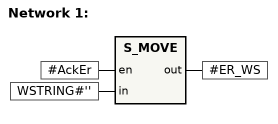
   IF #AckEr THEN #ER_WS := WSTRING#''; END_IF;
END_REGION

REGION Network 2 (SCL)

   #para_Artlimits := #para_in;
   #ER := false;
   IF #artLimfwd < #artLimRev THEN
       #ER_WS := #ER_WSlimfwdrev;
       #ER := true;
   ELSIF #UseArtLimitw THEN
       #para_Artlimits.pos_lim_fwd_USER := MIN(IN1 := #para_in.pos_lim_fwd_USER, IN2 := #artLimfwd);
       #para_Artlimits.pos_lim_rev_USER := MAX(IN1 := #para_in.pos_lim_rev_USER, IN2 := #artLimRev);
   END_IF;
END_REGION
END_FUNCTION_BLOCK

FUNCTION_BLOCK "axis_manager"   // FB25, FBD
{ S7_Optimized_Access := 'TRUE' }
VERSION : 0.1
// stored: AutoNumber true, IsIECCheckEnabled false, IsRetainMemResEnabled false, MemoryReserve 100, SetENOAutomatically false, UDAEnableTagReadback false
   VAR_INPUT
      allowed : Bool;
      targetUnison : Real;
      targetHome : Real;
      targetStep : Real;
      bSoftStop : Bool;
      bHome : Bool;
      hbStepPlus : Bool;
      hbStepMinus : Bool;
      bFwd : Bool;
      bRev : Bool;
      Params : "typeMotPara";
      ExecUni : Bool;
      theseAreDoors : Bool;
      xOverrideLOCAL : Bool;
      POS : Real;
   END_VAR
   VAR_OUTPUT
      team_unison : Bool;
      team_free : Bool;
      team_override : Bool;
      Desk_slowly : Bool;
      yaSpeedManual : Real;
      yaSpeedAuto : Real;
      m_auto : Bool;
      m_man : Bool;
      au_execute : Bool;
      aut_target : Real;
      OVERRIDE : Bool;
      ExecutingManuverFreeMode : Bool;
   END_VAR
   VAR
      st_Fwd : Bool;
      st_Rev : Bool;
      st_speed_slow_or_fast_negative : Real;
      aman_sel_target_Instance { S7_SetPoint := 'True'} : "aman_sel_target";
   END_VAR
   VAR_TEMP
      st_speedManual_slow_or_fast : Real;
      SpeedBlind : Real;
      stSpeedManualSlow : Real;
      Speed_autoSlow : Real;
   END_VAR
BEGIN

REGION Network 1
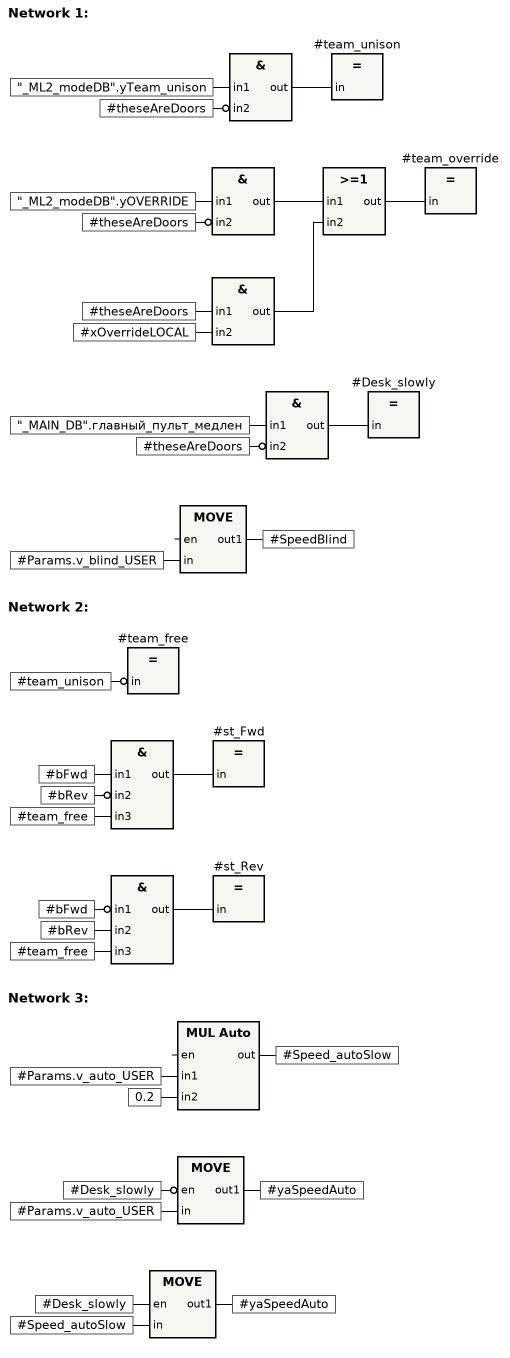
   #team_unison := "_ML2_modeDB".yTeam_unison AND NOT #theseAreDoors;
   #team_override := ("_ML2_modeDB".yOVERRIDE AND NOT #theseAreDoors) OR (#theseAreDoors AND #xOverrideLOCAL);
   #Desk_slowly := "_MAIN_DB".главный_пульт_медлен AND NOT #theseAreDoors;
   #SpeedBlind := #Params.v_blind_USER;
END_REGION

REGION Network 2
   #team_free := NOT #team_unison;
   #st_Fwd := #bFwd AND NOT #bRev AND #team_free;
   #st_Rev := NOT #bFwd AND #bRev AND #team_free;
END_REGION

REGION Network 3
   #Speed_autoSlow := #Params.v_auto_USER * 0.2;
   IF NOT #Desk_slowly THEN #yaSpeedAuto := #Params.v_auto_USER; END_IF;
   IF #Desk_slowly THEN #yaSpeedAuto := #Speed_autoSlow; END_IF;
END_REGION

REGION Network 4
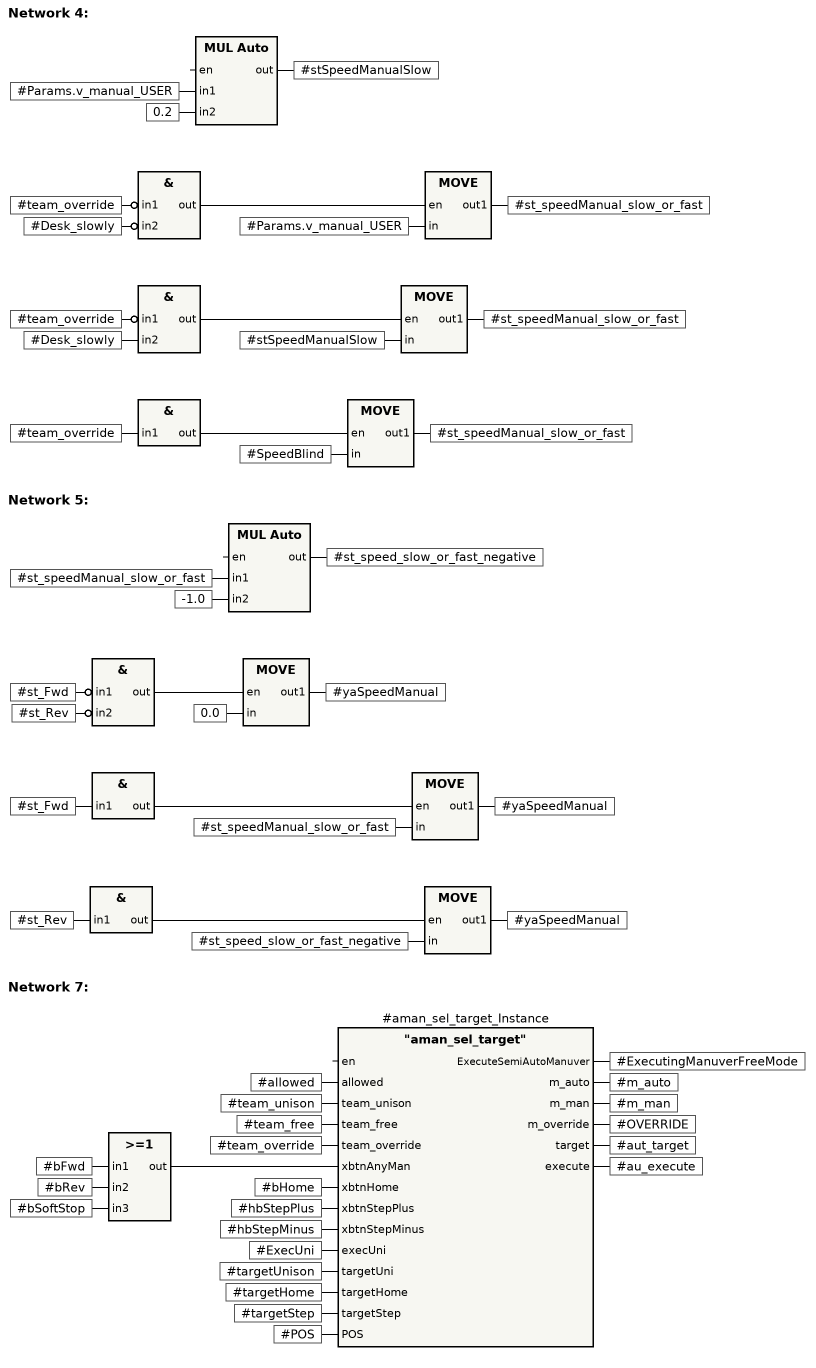
   #stSpeedManualSlow := #Params.v_manual_USER * 0.2;
   IF NOT #team_override AND NOT #Desk_slowly THEN
       #st_speedManual_slow_or_fast := #Params.v_manual_USER;
   END_IF;
   IF NOT #team_override AND #Desk_slowly THEN #st_speedManual_slow_or_fast := #stSpeedManualSlow; END_IF;
   IF #team_override THEN #st_speedManual_slow_or_fast := #SpeedBlind; END_IF;
END_REGION

REGION Network 5
   #st_speed_slow_or_fast_negative := #st_speedManual_slow_or_fast * (-1.0);
   IF NOT #st_Fwd AND NOT #st_Rev THEN #yaSpeedManual := 0.0; END_IF;
   IF #st_Fwd THEN #yaSpeedManual := #st_speedManual_slow_or_fast; END_IF;
   IF #st_Rev THEN #yaSpeedManual := #st_speed_slow_or_fast_negative; END_IF;
END_REGION

REGION Network 7
   #aman_sel_target_Instance(allowed := #allowed,   // "aman_sel_target"
                           team_unison := #team_unison,
                           team_free := #team_free,
                           team_override := #team_override,
                           xbtnAnyMan := #bFwd OR #bRev OR #bSoftStop,
                           xbtnHome := #bHome,
                           xbtnStepPlus := #hbStepPlus,
                           xbtnStepMinus := #hbStepMinus,
                           execUni := #ExecUni,
                           targetUni := #targetUnison,
                           targetHome := #targetHome,
                           targetStep := #targetStep,
                           POS := #POS,
                           ExecuteSemiAutoManuver => #ExecutingManuverFreeMode,
                           m_auto => #m_auto,
                           m_man => #m_man,
                           m_override => #OVERRIDE,
                           target => #aut_target,
                           execute => #au_execute);
END_REGION
END_FUNCTION_BLOCK

FUNCTION_BLOCK "aman_sel_target"   // FB58, FBD
{ S7_Optimized_Access := 'TRUE' }
VERSION : 0.1
// stored: AutoNumber true, IsIECCheckEnabled false, IsRetainMemResEnabled false, MemoryReserve 100, SetENOAutomatically false, UDAEnableTagReadback false
   VAR_INPUT
      allowed : Bool;
      team_unison : Bool;
      team_free : Bool;
      team_override : Bool;
      xbtnAnyMan : Bool;
      xbtnHome : Bool;
      xbtnStepPlus : Bool;
      xbtnStepMinus : Bool;
      execUni : Bool;
      targetUni : Real;
      targetHome : Real;
      targetStep : Real;
      POS : Real;
   END_VAR
   VAR_OUTPUT
      ExecuteSemiAutoManuver : Bool;
      m_auto : Bool;
      m_man : Bool;
      m_override : Bool;
      target : Real;
      execute : Bool;
   END_VAR
   VAR
      auto_allowed : Bool;
      anyBtn : Bool;
      xbtnHome_was : Bool;
      bsuhome { S7_SetPoint := 'True'} : "_ML2_ts_block1_subunit";
      p1Home : Bool;
      q1Home : Bool;
      Q_integer : Int;
      bsu_step_plus { S7_SetPoint := 'True'} : "_ML2_ts_block1_subunit";
      p2StepPlus : Bool;
      q2StepPlus : Bool;
      p3StepMinus : Bool;
      q3StepMinus : Bool;
      bsu_step_minus { S7_SetPoint := 'True'} : "_ML2_ts_block1_subunit";
   END_VAR
   VAR CONSTANT
      Qi0_off : Int := 0;
      Qi1_home : Int := 1;
      Qi2_stepPlus : Int := 2;
      Qi3_stepMinus : Int := 3;
   END_VAR
BEGIN

REGION Network 1
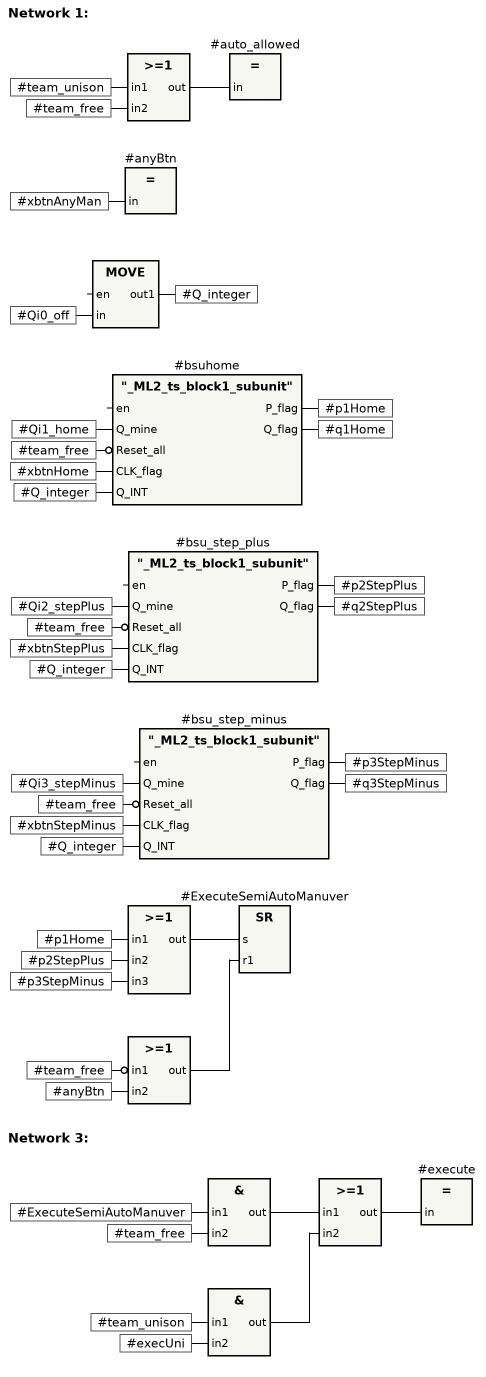
   #auto_allowed := #team_unison OR #team_free;
   #anyBtn := #xbtnAnyMan;
   #Q_integer := #Qi0_off;
   #bsuhome(Q_mine := #Qi1_home,   // "_ML2_ts_block1_subunit"
            Reset_all := NOT #team_free,
            CLK_flag := #xbtnHome,
            Q_INT := #Q_integer,
            P_flag => #p1Home,
            Q_flag => #q1Home);
   #bsu_step_plus(Q_mine := #Qi2_stepPlus,   // "_ML2_ts_block1_subunit"
                  Reset_all := NOT #team_free,
                  CLK_flag := #xbtnStepPlus,
                  Q_INT := #Q_integer,
                  P_flag => #p2StepPlus,
                  Q_flag => #q2StepPlus);
   #bsu_step_minus(Q_mine := #Qi3_stepMinus,   // "_ML2_ts_block1_subunit"
                   Reset_all := NOT #team_free,
                   CLK_flag := #xbtnStepMinus,
                   Q_INT := #Q_integer,
                   P_flag => #p3StepMinus,
                   Q_flag => #q3StepMinus);
   IF #p1Home OR #p2StepPlus OR #p3StepMinus THEN
       #ExecuteSemiAutoManuver := TRUE;   // SR flip-flop
   END_IF;
   IF NOT #team_free OR #anyBtn THEN #ExecuteSemiAutoManuver := FALSE; END_IF;
END_REGION

REGION Network 2 (SCL)
   IF #p1Home THEN
       #target := #targetHome;
   ELSIF #p2StepPlus THEN
       #target := #POS + #targetStep;
   ELSIF #p3StepMinus THEN
       #target := #POS - #targetStep;
   ELSIF #team_unison THEN
       #target := #targetUni;
   END_IF;
   #xbtnHome_was := #xbtnHome;
END_REGION

REGION Network 3
   #execute := (#ExecuteSemiAutoManuver AND #team_free) OR (#team_unison AND #execUni);
END_REGION

REGION Network 4
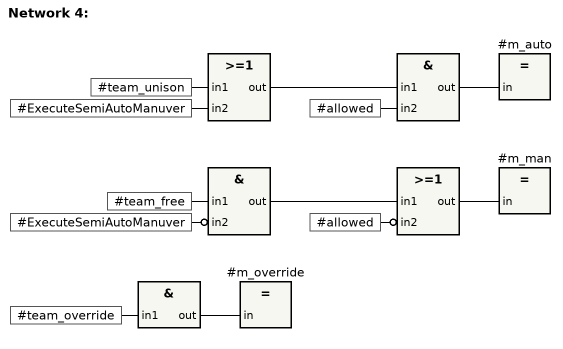
   #m_auto := (#team_unison OR #ExecuteSemiAutoManuver) AND #allowed;
   #m_man := (#team_free AND NOT #ExecuteSemiAutoManuver) OR NOT #allowed;
   #m_override := #team_override;
END_REGION
END_FUNCTION_BLOCK

FUNCTION_BLOCK "__mot_universal_"   // FB18, FBD
{ S7_Optimized_Access := 'TRUE' }
VERSION : 0.1
// stored: AutoNumber true, IsIECCheckEnabled false, IsRetainMemResEnabled false, MemoryReserve 100, SetENOAutomatically false, UDAEnableTagReadback false
   VAR_INPUT
      ALLOWED : Bool;
      ALLOWED_ONLY_IN_OVERRIDE : Bool;
      OVERRIDE_NOW : Bool;
      isMultiturn : Bool;
      MultiTurnGoesFwdOnly : Bool;
      xFwdOk : Bool;
      xRevOk : Bool;
      xPredefCal : Bool;
      MAN_SET_SPEED_maxParSpeed : Real;
      ENC : Real;
      par : "typeMotPara";
      partnerCalibrated : Bool := true;
      artLimits : Bool;
      artLimFwd : Real;
      artLimRev : Real;
      AU_EXECUTE_TO_TARGET : Bool;
      AU_SPD : Real;
      AUT_MD_SPD_notPos : Bool := false;
      AUT : Bool;
      MAN : Bool;
      CLOCK_S_P_SCAN { ExternalWritable := 'False'} : Real;
      ALIEN_HOST_CONTROL_MODE_ENABLE : Bool;
      ALIEN_FWD : Bool;
      ALIEN_REV : Bool;
      ALIEN_SPEED_ABS : Real;
      TheseAreDoors : Bool;
   END_VAR
   VAR_OUTPUT
      AU_INPOS : Bool;
      FWD : Bool;
      REV : Bool;
      BRK_REL : Bool;
      SPEED_ABS : Real;
      SPEED : Real;
      BLIND : Bool;
      ER_FOLLOW : Bool;
      ER_SET : Bool;
      ER_FWD : Bool;
      ER_REV : Bool;
      er_ws : WString;
   END_VAR
   VAR_IN_OUT
      AU_TRGT : Real;
      calibrated : Bool;
      POS : Real;
      ENC_RET_DATA : "typePOSMEMcalib";
   END_VAR
   VAR
      par_Local : "typeMotPara";
      SERV_block : Bool;
      AUTO_static : Bool;
      MAN_static : Bool := TRUE;
      M_MD { S7_SetPoint := 'True'} : "MD";
      ENC_DB { S7_SetPoint := 'True'} : "encoder";
      manual { S7_SetPoint := 'True'} : "manual_analog";
      auto { S7_SetPoint := 'True'} : "auto_analog_NORMAL";
      ENC_CHECK { S7_SetPoint := 'True'} : "enc_no_change_in_time";
      BRK_DB { S7_SetPoint := 'True'} : "BRK_FB";
      sr_auto { S7_SetPoint := 'True'} : "SR_TRIG";
      sr_man { S7_SetPoint := 'True'} : "SR_TRIG";
      auto_analog_Speed_Instance { S7_SetPoint := 'True'} : "auto_analog_copySpeed";
      speed_slowed_by_inertia : Real;
      speed_command : Real;
      mot_speed_wdir_slowly_accelerated_Instance { S7_SetPoint := 'True'} : "mot_speed_wdir_slowly_accelerated";
      mot_missed_target { S7_SetPoint := 'True'} : "mot_universal_arrived_missed";
      arrived_missed : Bool;
   END_VAR
   VAR_TEMP
      reset_y : Bool;
      BRK_NOW_ERROR_EXISTS : Bool;
      speed_fast_neg : Real;
      placeHolderreal : Real;
      er_set_1m : Bool;
      er_set_1a1 : Bool;
      er_set_1a2 : Bool;
      er_set_2 : Bool;
      er_set_3 : Bool;
      inertia_Mode : Bool;
      erws1m0 : WString;
      erws1a1 : WString;
      erws1a2 : WString;
      erws2 : WString;
      erws3 : WString;
   END_VAR
   VAR CONSTANT
      erwsNOER : WString := WSTRING#'no er';
   END_VAR
BEGIN

REGION Network 1
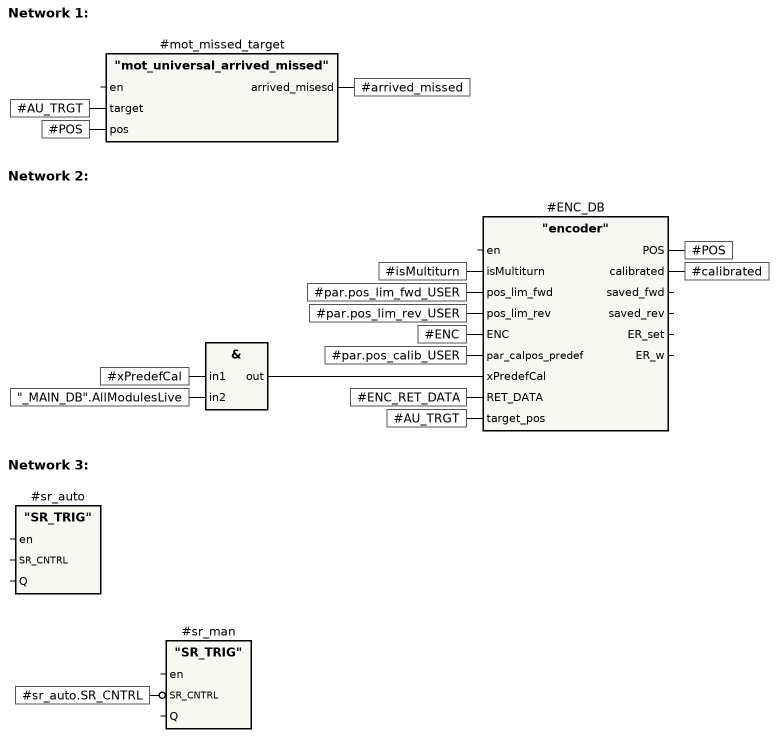
   #mot_missed_target(target := #AU_TRGT, pos := #POS, arrived_misesd => #arrived_missed);   // "mot_universal_arrived_missed"
END_REGION

REGION Network 2
   #ENC_DB(isMultiturn := #isMultiturn,   // "encoder"
           pos_lim_fwd := #par.pos_lim_fwd_USER,
           pos_lim_rev := #par.pos_lim_rev_USER,
           ENC := #ENC,
           par_calpos_predef := #par.pos_calib_USER,
           xPredefCal := #xPredefCal AND "_MAIN_DB".AllModulesLive,
           RET_DATA := #ENC_RET_DATA,
           target_pos := #AU_TRGT,
           POS => #POS,
           calibrated => #calibrated);
END_REGION

REGION Network 3
   #sr_auto();   // "SR_TRIG"
   #sr_man(SR_CNTRL := NOT #sr_auto.SR_CNTRL);   // "SR_TRIG"
END_REGION

REGION Network 4 (SCL)
   #SERV_block := #ALIEN_HOST_CONTROL_MODE_ENABLE;
   IF #SERV_block THEN
       #FWD := #ALIEN_FWD;
       #REV := #ALIEN_REV;
       #SPEED_ABS := #ALIEN_SPEED_ABS;
   END_IF;
END_REGION

REGION Network 5
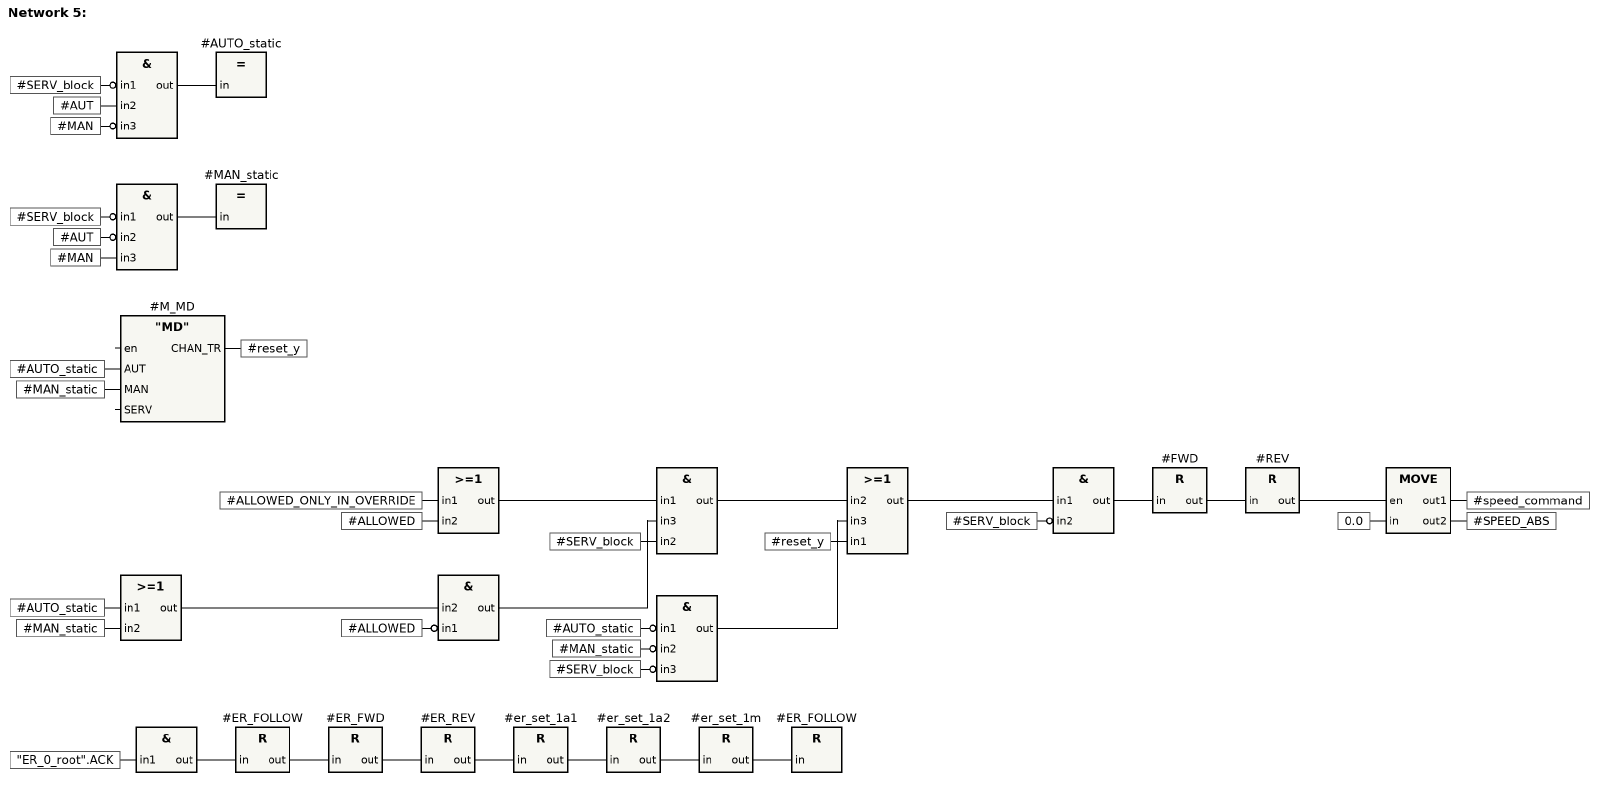
   #AUTO_static := NOT #SERV_block AND #AUT AND NOT #MAN;
   #MAN_static := NOT #SERV_block AND NOT #AUT AND #MAN;
   #M_MD(AUT := #AUTO_static, MAN := #MAN_static, CHAN_TR => #reset_y);   // "MD"
   IF (((#ALLOWED_ONLY_IN_OVERRIDE OR #ALLOWED) AND (#AUTO_static OR #MAN_static) AND NOT #ALLOWED AND #SERV_block) OR (NOT #AUTO_static AND NOT #MAN_static AND NOT #SERV_block) OR #reset_y) AND NOT #SERV_block THEN
       #FWD := FALSE;
       #REV := FALSE;
       #speed_command := 0.0;
       #SPEED_ABS := 0.0;
   END_IF;
   IF "ER_0_root".ACK THEN
       #ER_FOLLOW := FALSE;
       #ER_FWD := FALSE;
       #ER_REV := FALSE;
       #er_set_1a1 := FALSE;
       #er_set_1a2 := FALSE;
       #er_set_1m := FALSE;
       #ER_FOLLOW := FALSE;
   END_IF;
END_REGION

REGION Network 6
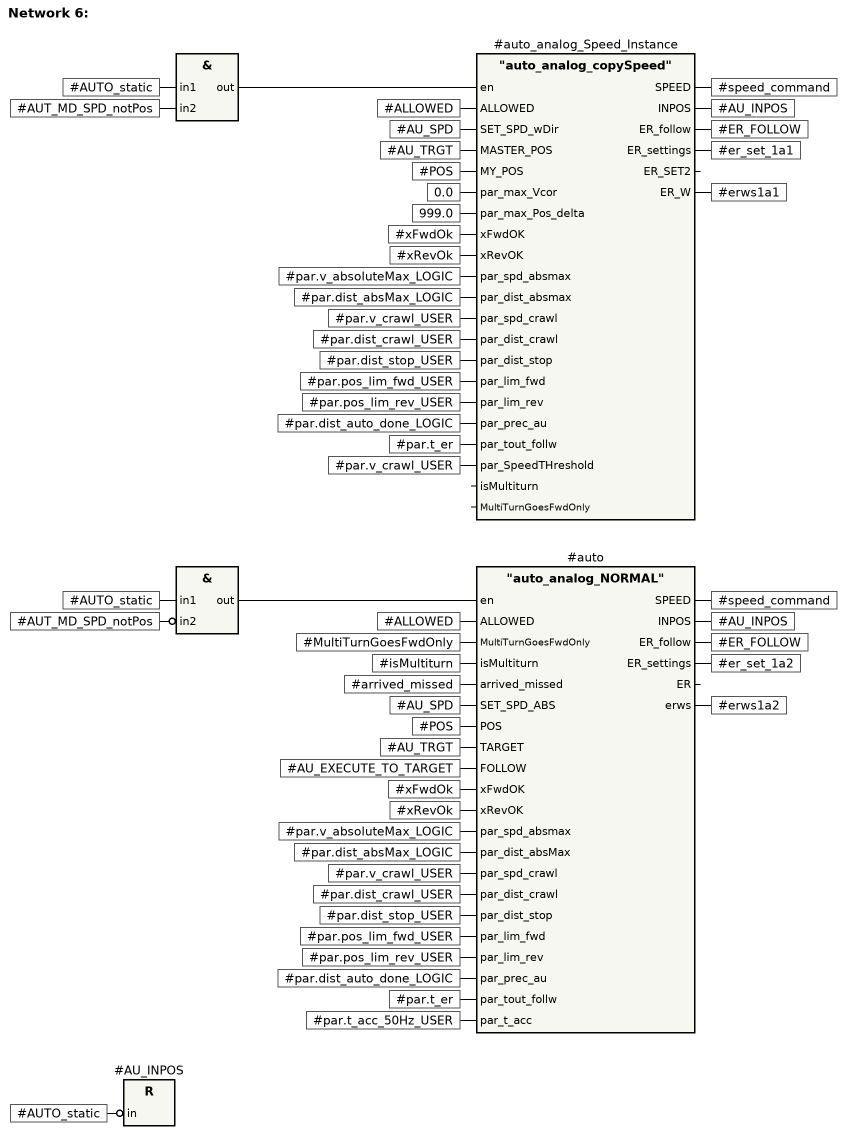
   IF #AUTO_static AND #AUT_MD_SPD_notPos THEN
       #auto_analog_Speed_Instance(ALLOWED := #ALLOWED,   // "auto_analog_copySpeed"
                               SET_SPD_wDir := #AU_SPD,
                               MASTER_POS := #AU_TRGT,
                               MY_POS := #POS,
                               par_max_Vcor := 0.0,
                               par_max_Pos_delta := 999.0,
                               xFwdOK := #xFwdOk,
                               xRevOK := #xRevOk,
                               par_spd_absmax := #par.v_absoluteMax_LOGIC,
                               par_dist_absmax := #par.dist_absMax_LOGIC,
                               par_spd_crawl := #par.v_crawl_USER,
                               par_dist_crawl := #par.dist_crawl_USER,
                               par_dist_stop := #par.dist_stop_USER,
                               par_lim_fwd := #par.pos_lim_fwd_USER,
                               par_lim_rev := #par.pos_lim_rev_USER,
                               par_prec_au := #par.dist_auto_done_LOGIC,
                               par_tout_follw := #par.t_er,
                               par_SpeedTHreshold := #par.v_crawl_USER,
                               SPEED => #speed_command,
                               INPOS => #AU_INPOS,
                               ER_follow => #ER_FOLLOW,
                               ER_settings => #er_set_1a1,
                               ER_W => #erws1a1);
   END_IF;
   IF #AUTO_static AND NOT #AUT_MD_SPD_notPos THEN
       #auto(ALLOWED := #ALLOWED,   // "auto_analog_NORMAL"
             MultiTurnGoesFwdOnly := #MultiTurnGoesFwdOnly,
             isMultiturn := #isMultiturn,
             arrived_missed := #arrived_missed,
             SET_SPD_ABS := #AU_SPD,
             POS := #POS,
             TARGET := #AU_TRGT,
             FOLLOW := #AU_EXECUTE_TO_TARGET,
             xFwdOK := #xFwdOk,
             xRevOK := #xRevOk,
             par_spd_absmax := #par.v_absoluteMax_LOGIC,
             par_dist_absMax := #par.dist_absMax_LOGIC,
             par_spd_crawl := #par.v_crawl_USER,
             par_dist_crawl := #par.dist_crawl_USER,
             par_dist_stop := #par.dist_stop_USER,
             par_lim_fwd := #par.pos_lim_fwd_USER,
             par_lim_rev := #par.pos_lim_rev_USER,
             par_prec_au := #par.dist_auto_done_LOGIC,
             par_tout_follw := #par.t_er,
             par_t_acc := #par.t_acc_50Hz_USER,
             SPEED => #speed_command,
             INPOS => #AU_INPOS,
             ER_follow => #ER_FOLLOW,
             ER_settings => #er_set_1a2,
             erws => #erws1a2);
   END_IF;
   IF NOT #AUTO_static THEN #AU_INPOS := FALSE; END_IF;
END_REGION

REGION Network 7 (SCL)

   //#MAN_SET_SPEED_maxParSpeed := #MAN_SET_SPEED_maxParSpeed;
END_REGION

REGION Network 8
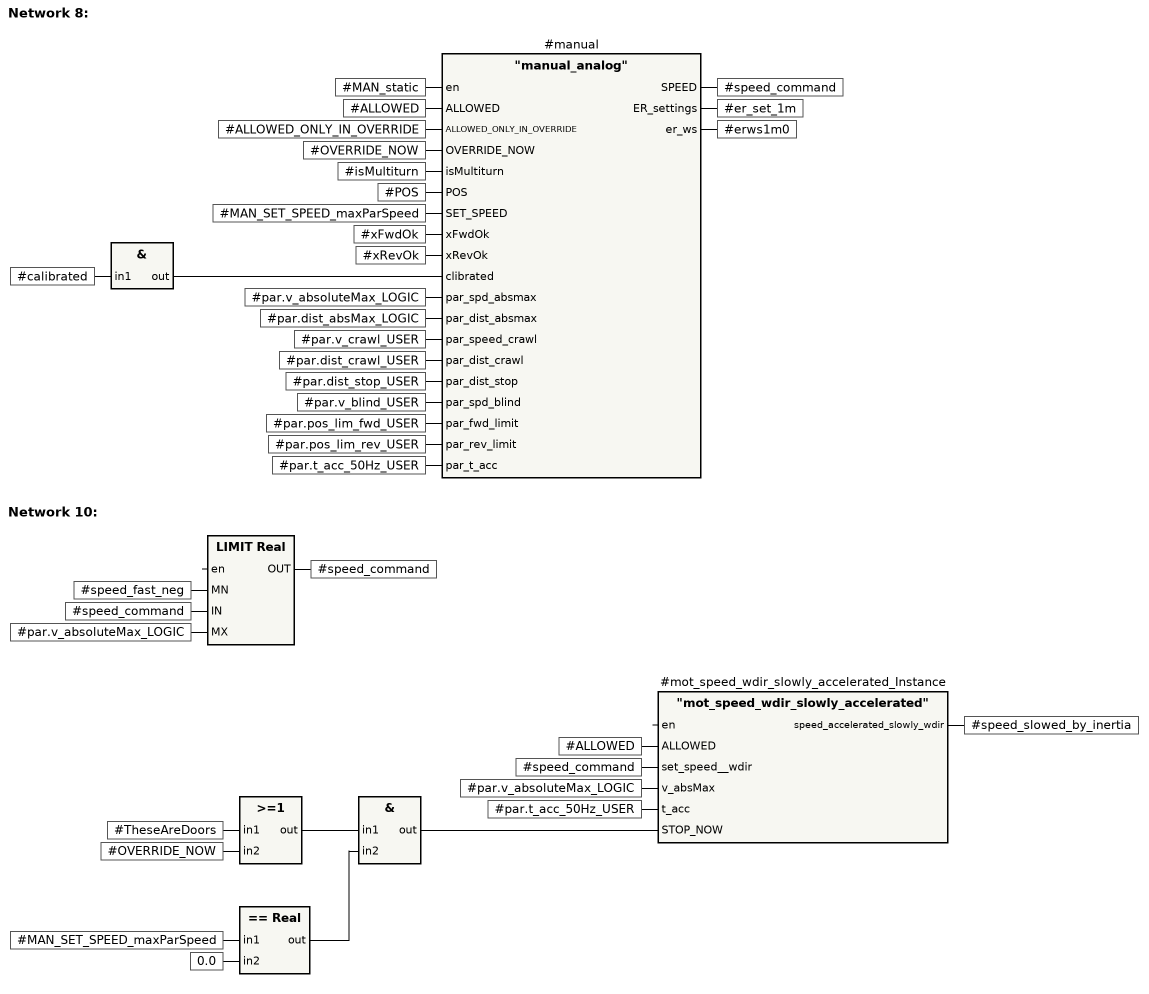
   IF #MAN_static THEN
       #manual(ALLOWED := #ALLOWED,   // "manual_analog"
               ALLOWED_ONLY_IN_OVERRIDE := #ALLOWED_ONLY_IN_OVERRIDE,
               OVERRIDE_NOW := #OVERRIDE_NOW,
               isMultiturn := #isMultiturn,
               POS := #POS,
               SET_SPEED := #MAN_SET_SPEED_maxParSpeed,
               xFwdOk := #xFwdOk,
               xRevOk := #xRevOk,
               clibrated := #calibrated,
               par_spd_absmax := #par.v_absoluteMax_LOGIC,
               par_dist_absmax := #par.dist_absMax_LOGIC,
               par_speed_crawl := #par.v_crawl_USER,
               par_dist_crawl := #par.dist_crawl_USER,
               par_dist_stop := #par.dist_stop_USER,
               par_spd_blind := #par.v_blind_USER,
               par_fwd_limit := #par.pos_lim_fwd_USER,
               par_rev_limit := #par.pos_lim_rev_USER,
               par_t_acc := #par.t_acc_50Hz_USER,
               SPEED => #speed_command,
               ER_settings => #er_set_1m,
               er_ws => #erws1m0);
   END_IF;
END_REGION

REGION Network 9 (SCL)
   #speed_fast_neg := -#par.v_absoluteMax_LOGIC;
END_REGION

REGION Network 10
   #speed_command := LIMIT(MN := #speed_fast_neg, IN := #speed_command, MX := #par.v_absoluteMax_LOGIC);
   #mot_speed_wdir_slowly_accelerated_Instance(ALLOWED := #ALLOWED,   // "mot_speed_wdir_slowly_accelerated"
                           set_speed__wdir := #speed_command,
                           v_absMax := #par.v_absoluteMax_LOGIC,
                           t_acc := #par.t_acc_50Hz_USER,
                           STOP_NOW := (#TheseAreDoors OR #OVERRIDE_NOW) AND (#MAN_SET_SPEED_maxParSpeed = 0.0),
                           speed_accelerated_slowly_wdir => #speed_slowed_by_inertia);
END_REGION

REGION Network 11 (SCL)
   IF NOT #SERV_block THEN
       #FWD := #speed_slowed_by_inertia > 0;
       #REV := #speed_slowed_by_inertia < 0;
   END_IF;
END_REGION

REGION Network 12
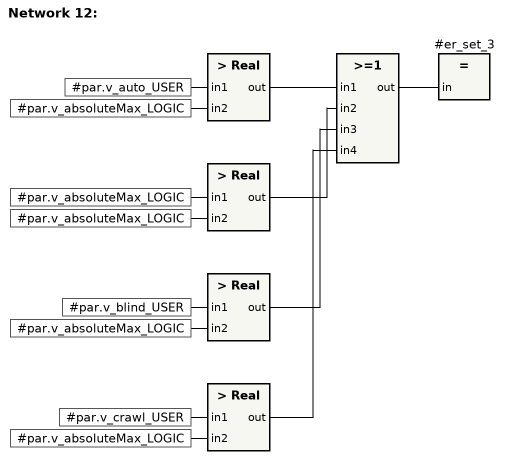
   #er_set_3 := (#par.v_auto_USER > #par.v_absoluteMax_LOGIC) OR (#par.v_absoluteMax_LOGIC > #par.v_absoluteMax_LOGIC) OR (#par.v_blind_USER > #par.v_absoluteMax_LOGIC) OR (#par.v_crawl_USER > #par.v_absoluteMax_LOGIC);
END_REGION

REGION Network 13
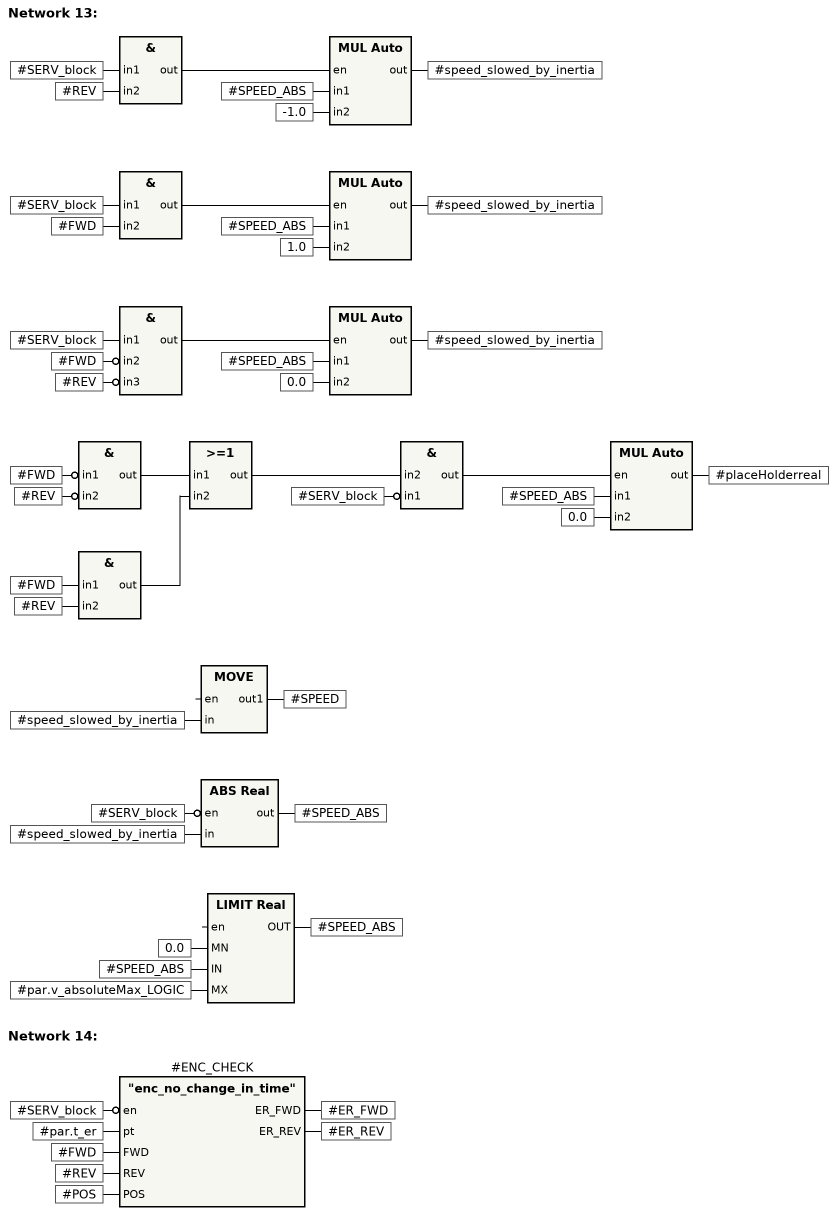
   IF #SERV_block AND #REV THEN #speed_slowed_by_inertia := #SPEED_ABS * (-1.0); END_IF;
   IF #SERV_block AND #FWD THEN #speed_slowed_by_inertia := #SPEED_ABS * 1.0; END_IF;
   IF #SERV_block AND NOT #FWD AND NOT #REV THEN #speed_slowed_by_inertia := #SPEED_ABS * 0.0; END_IF;
   IF ((NOT #FWD AND NOT #REV) OR (#FWD AND #REV)) AND NOT #SERV_block THEN
       #placeHolderreal := #SPEED_ABS * 0.0;
   END_IF;
   #SPEED := #speed_slowed_by_inertia;
   IF NOT #SERV_block THEN #SPEED_ABS := ABS(#speed_slowed_by_inertia); END_IF;
   #SPEED_ABS := LIMIT(MN := 0.0, IN := #SPEED_ABS, MX := #par.v_absoluteMax_LOGIC);
END_REGION

REGION Network 14
   IF NOT #SERV_block THEN
       #ENC_CHECK(pt := #par.t_er, FWD := #FWD, REV := #REV, POS := #POS, ER_FWD => #ER_FWD, ER_REV => #ER_REV);   // "enc_no_change_in_time"
   END_IF;
END_REGION

REGION Network 15
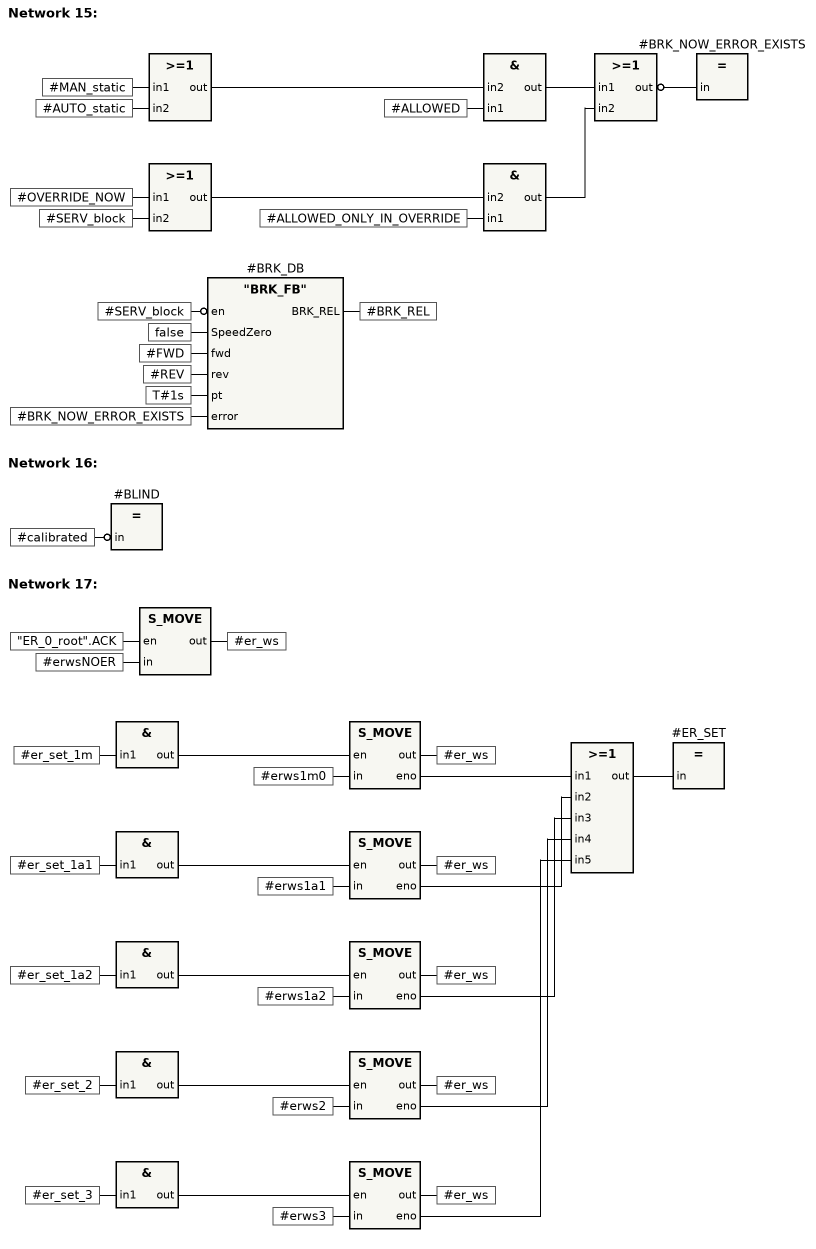
   #BRK_NOW_ERROR_EXISTS := NOT (((#MAN_static OR #AUTO_static) AND #ALLOWED) OR ((#OVERRIDE_NOW OR #SERV_block) AND #ALLOWED_ONLY_IN_OVERRIDE));
   IF NOT #SERV_block THEN
       #BRK_DB(SpeedZero := false,   // "BRK_FB"
               fwd := #FWD,
               rev := #REV,
               pt := T#1s,
               error := #BRK_NOW_ERROR_EXISTS,
               BRK_REL => #BRK_REL);
   END_IF;
END_REGION

REGION Network 16
   #BLIND := NOT #calibrated;
END_REGION

REGION Network 17
   IF "ER_0_root".ACK THEN #er_ws := #erwsNOER; END_IF;
   IF #er_set_1m THEN #er_ws := #erws1m0; END_IF;
   IF #er_set_1a1 THEN #er_ws := #erws1a1; END_IF;
   IF #er_set_1a2 THEN #er_ws := #erws1a2; END_IF;
   IF #er_set_2 THEN #er_ws := #erws2; END_IF;
   IF #er_set_3 THEN #er_ws := #erws3; END_IF;
   #ER_SET := #er_set_1m OR #er_set_1a1 OR #er_set_1a2 OR #er_set_2 OR #er_set_3;
END_REGION
END_FUNCTION_BLOCK

FUNCTION_BLOCK "encoder"   // FB15, FBD
{ S7_Optimized_Access := 'TRUE' }
VERSION : 0.1
// stored: AutoNumber true, IsIECCheckEnabled false, IsRetainMemResEnabled false, MemoryReserve 100, SetENOAutomatically false, UDAEnableTagReadback false
   VAR_INPUT
      isMultiturn : Bool;
      pos_lim_fwd : Real;
      pos_lim_rev : Real;
      ENC : Real;
      par_calpos_predef : Real;
      xPredefCal : Bool;
   END_VAR
   VAR_OUTPUT
      POS : Real;
      calibrated : Bool;
      saved_fwd : Real;
      saved_rev : Real;
      ER_set : Bool;
      ER_w : WString;
   END_VAR
   VAR_IN_OUT
      RET_DATA : "typePOSMEMcalib";
      target_pos : Real;
   END_VAR
   VAR
      not_first_scan : Bool;
      xPredefCal_filtered : Bool;
      tr_predef : R_TRIG;
      tr_fwd : R_TRIG;
      tr_rev : R_TRIG;
      ton_filter { S7_SetPoint := 'True'} : TON_TIME;
   END_VAR
   VAR_TEMP
      btn_calib_now_predef : Bool;
      btn_calib_now_fwd : Bool;
      btn_calib_now_rev : Bool;
      length_rev_fwd : Real;
   END_VAR
BEGIN

REGION Network 1
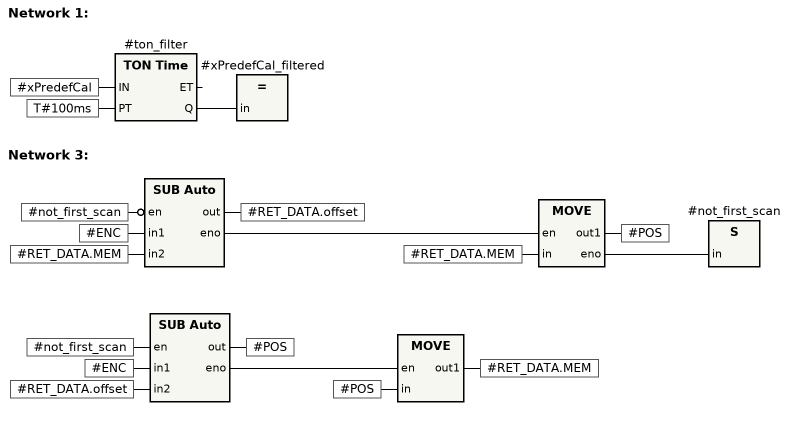
   #ton_filter(IN := #xPredefCal, PT := T#100ms);   // TON
   #xPredefCal_filtered := #ton_filter.Q;
END_REGION

REGION Network 2 (SCL)
   IF #isMultiturn THEN
       IF NOT #RET_DATA.calibrated THEN
           #RET_DATA.calibrated := true;
       END_IF;
       IF #pos_lim_fwd > #pos_lim_rev THEN
           #ER_set := false;
           #ER_w := WString#'';
           #length_rev_fwd := #pos_lim_fwd - #pos_lim_rev;
           IF #POS >= #pos_lim_fwd THEN


               #RET_DATA.offset := #RET_DATA.offset + #length_rev_fwd;
           END_IF;
           IF #POS < #pos_lim_rev THEN
               #RET_DATA.offset := #RET_DATA.offset - #length_rev_fwd;
           END_IF;



           IF #target_pos >= #pos_lim_fwd THEN
               #target_pos := #target_pos - #length_rev_fwd;
           END_IF;
           IF #target_pos < #pos_lim_rev THEN
               #target_pos := #target_pos + #length_rev_fwd;
           END_IF;
       ELSE
           #ER_set := true;
           #ER_w := WString#'enc_fwd_lt_rev';
       END_IF;
   END_IF;
END_REGION

REGION Network 3
   IF NOT #not_first_scan THEN
       #RET_DATA.offset := #ENC - #RET_DATA.MEM;
       #POS := #RET_DATA.MEM;
       #not_first_scan := TRUE;
   END_IF;
   IF #not_first_scan THEN
       #POS := #ENC - #RET_DATA.offset;
       #RET_DATA.MEM := #POS;
   END_IF;
END_REGION

REGION Network 4 (SCL)
   #tr_predef(CLK := #xPredefCal_filtered);

   #btn_calib_now_predef := #tr_predef.Q;

   IF #btn_calib_now_predef THEN
       #RET_DATA.offset := #ENC - #par_calpos_predef;
       #RET_DATA.calibrated := true;
   END_IF;

   #calibrated := #RET_DATA.calibrated;
END_REGION
END_FUNCTION_BLOCK

FUNCTION_BLOCK "SR_TRIG"   // FB34, FBD
{ S7_Optimized_Access := 'TRUE' }
VERSION : 0.1
// stored: AutoNumber true, IsIECCheckEnabled false, IsRetainMemResEnabled false, MemoryReserve 100, SetENOAutomatically false, UDAEnableTagReadback false
   VAR_INPUT
      SR_CNTRL : Bool;
   END_VAR
   VAR_IN_OUT
      Q : Bool;
   END_VAR
   VAR
      mem1 : Bool;
      mem2 : Bool;
   END_VAR
   VAR_TEMP   // added for the SCL form of the ladder/FBD networks
      _w1 : Bool;
      _w2 : Bool;
   END_VAR
BEGIN

REGION Network 1
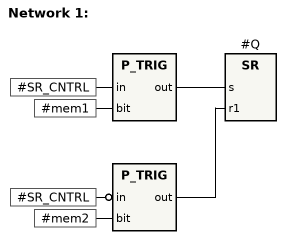
   #_w1 := #SR_CNTRL AND NOT #mem1;   // rising edge
   #mem1 := #SR_CNTRL;
   #_w2 := NOT #SR_CNTRL AND NOT #mem2;   // rising edge
   #mem2 := NOT #SR_CNTRL;
   IF #_w1 THEN
       #Q := TRUE;   // SR flip-flop
   END_IF;
   IF #_w2 THEN #Q := FALSE; END_IF;
END_REGION
END_FUNCTION_BLOCK

FUNCTION_BLOCK "MD"   // FB11, FBD
{ S7_Optimized_Access := 'TRUE' }
VERSION : 0.1
// stored: AutoNumber true, IsIECCheckEnabled false, IsRetainMemResEnabled false, MemoryReserve 100, SetENOAutomatically false, UDAEnableTagReadback false
   VAR_OUTPUT
      CHAN_TR : Bool;
   END_VAR
   VAR_IN_OUT
      AUT : Bool;
      MAN : Bool := true;
      SERV : Bool;
   END_VAR
   VAR
      lbs { S7_SetPoint := 'True'} : "last_button_stands";
   END_VAR
BEGIN

REGION Network 1
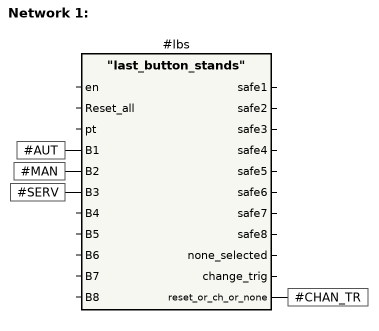
   #lbs(B1 := #AUT, B2 := #MAN, B3 := #SERV, reset_or_ch_or_none => #CHAN_TR);   // "last_button_stands"
END_REGION
END_FUNCTION_BLOCK

FUNCTION_BLOCK "auto_analog_copySpeed"   // FB22, FBD
{ S7_Optimized_Access := 'TRUE' }
VERSION : 0.1
// stored: AutoNumber true, IsIECCheckEnabled false, IsRetainMemResEnabled false, MemoryReserve 100, SetENOAutomatically false, UDAEnableTagReadback false
   VAR_INPUT
      ALLOWED : Bool;
      SET_SPD_wDir { ExternalAccessible := 'False'; ExternalVisible := 'False'; ExternalWritable := 'False'} : Real;
      MASTER_POS : Real;
      MY_POS : Real;
      par_max_Vcor : Real;
      par_max_Pos_delta : Real;
      xFwdOK : Bool;
      xRevOK : Bool;
      par_spd_absmax : Real;
      par_dist_absmax : Real;
      par_spd_crawl : Real;
      par_dist_crawl : Real;
      par_dist_stop : Real;
      par_lim_fwd : Real;
      par_lim_rev : Real;
      par_prec_au : Real;
      par_tout_follw : Time;
      par_SpeedTHreshold : Real;
      isMultiturn : Bool;
      MultiTurnGoesFwdOnly : Bool;
   END_VAR
   VAR_OUTPUT
      SPEED : Real;
      INPOS : Bool;
      ER_follow : Bool;
      ER_settings : Bool;
      ER_SET2 : Bool;
      ER_W : WString;
   END_VAR
   VAR
      should_move_static : Bool;
   END_VAR
   VAR_TEMP
      dir_fwd : Bool;
      dir_rev : Bool;
      arrived : Bool;
      distance : Real;
      estop_ok_no_err : Bool;
      speed_by_lag : Real;
      speed_by_lag_pos : Real;
      speed_out_abs : Real;
      xFWDREV_matter : Bool;
      limits_matter : Bool;
   END_VAR
BEGIN

REGION Network 2
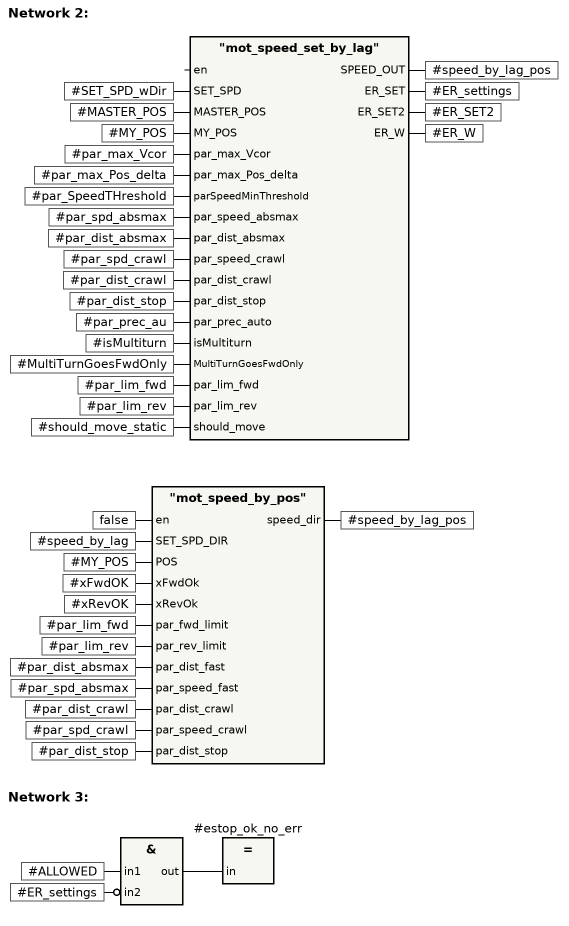
   "mot_speed_set_by_lag"(SET_SPD := #SET_SPD_wDir,
                          MASTER_POS := #MASTER_POS,
                          MY_POS := #MY_POS,
                          par_max_Vcor := #par_max_Vcor,
                          par_max_Pos_delta := #par_max_Pos_delta,
                          parSpeedMinThreshold := #par_SpeedTHreshold,
                          par_speed_absmax := #par_spd_absmax,
                          par_dist_absmax := #par_dist_absmax,
                          par_speed_crawl := #par_spd_crawl,
                          par_dist_crawl := #par_dist_crawl,
                          par_dist_stop := #par_dist_stop,
                          par_prec_auto := #par_prec_au,
                          isMultiturn := #isMultiturn,
                          MultiTurnGoesFwdOnly := #MultiTurnGoesFwdOnly,
                          par_lim_fwd := #par_lim_fwd,
                          par_lim_rev := #par_lim_rev,
                          should_move := #should_move_static,
                          SPEED_OUT => #speed_by_lag_pos,
                          ER_SET => #ER_settings,
                          ER_SET2 => #ER_SET2,
                          ER_W => #ER_W);
   IF false THEN
       "mot_speed_by_pos"(SET_SPD_DIR := #speed_by_lag,
                          POS := #MY_POS,
                          xFwdOk := #xFwdOK,
                          xRevOk := #xRevOK,
                          par_fwd_limit := #par_lim_fwd,
                          par_rev_limit := #par_lim_rev,
                          par_dist_fast := #par_dist_absmax,
                          par_speed_fast := #par_spd_absmax,
                          par_dist_crawl := #par_dist_crawl,
                          par_speed_crawl := #par_spd_crawl,
                          par_dist_stop := #par_dist_stop,
                          speed_dir => #speed_by_lag_pos);
   END_IF;
END_REGION

REGION Network 3
   #estop_ok_no_err := #ALLOWED AND NOT #ER_settings;
END_REGION

REGION Network 4 (SCL)
   #INPOS := ABS(#MASTER_POS - #MY_POS) < #par_prec_au;
END_REGION

REGION Network 5
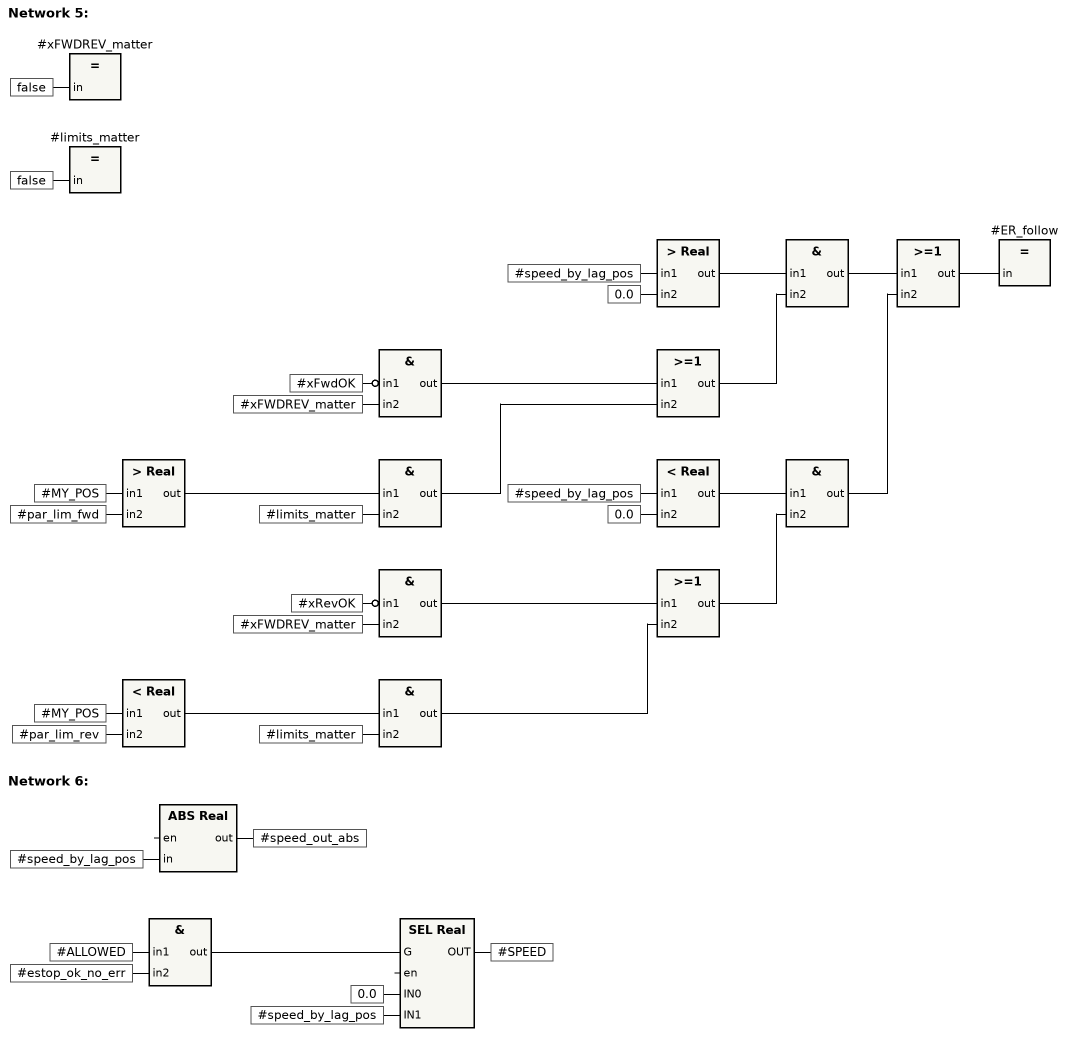
   #xFWDREV_matter := false;
   #limits_matter := false;
   #ER_follow := ((#speed_by_lag_pos > 0.0) AND ((NOT #xFwdOK AND #xFWDREV_matter) OR ((#MY_POS > #par_lim_fwd) AND #limits_matter))) OR ((#speed_by_lag_pos < 0.0) AND ((NOT #xRevOK AND #xFWDREV_matter) OR ((#MY_POS < #par_lim_rev) AND #limits_matter)));
END_REGION

REGION Network 6
   #speed_out_abs := ABS(#speed_by_lag_pos);
   #SPEED := SEL(G := #ALLOWED AND #estop_ok_no_err, IN0 := 0.0, IN1 := #speed_by_lag_pos);
END_REGION
END_FUNCTION_BLOCK

FUNCTION "mot_speed_set_by_lag" : Void   // FC5, FBD
{ S7_Optimized_Access := 'TRUE' }
VERSION : 0.1
// stored: AutoNumber true, IsIECCheckEnabled false, SetENOAutomatically false, UDAEnableTagReadback false
   VAR_INPUT
      SET_SPD : Real;
      MASTER_POS : Real;
      MY_POS : Real;
      par_max_Vcor : Real;
      par_max_Pos_delta : Real;
      parSpeedMinThreshold : Real;
      par_speed_absmax : Real;
      par_dist_absmax : Real;
      par_speed_crawl : Real;
      par_dist_crawl : Real;
      par_dist_stop : Real;
      par_prec_auto : Real;
      isMultiturn : Bool;
      MultiTurnGoesFwdOnly : Bool;
      par_lim_fwd : Real;
      par_lim_rev : Real;
   END_VAR
   VAR_OUTPUT
      SPEED_OUT : Real;
      ER_SET : Bool;
      ER_SET2 : Bool;
      ER_W : WString;
   END_VAR
   VAR_IN_OUT
      should_move : Bool;
   END_VAR
   VAR_TEMP
      delta_pos : Real;
      speed_cor : Real;
      scaled_delta_pos : Real;
      temp_speed : Real;
      speed_target : Real;
      set_speed_substantial : Bool;
      in_vicinity : Bool;
      delta : Real;
      set_speed_miniscule : Bool;
      SET_SPD_ABS : Real;
   END_VAR
BEGIN

REGION Network 1
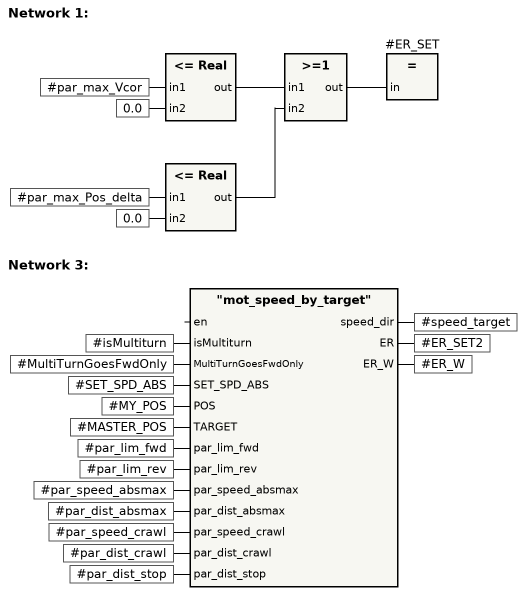
   #ER_SET := (#par_max_Vcor <= 0.0) OR (#par_max_Pos_delta <= 0.0);
END_REGION

REGION Network 2 (SCL)
   #SET_SPD_ABS := ABS(#SET_SPD);
END_REGION

REGION Network 3
   "mot_speed_by_target"(isMultiturn := #isMultiturn,
                         MultiTurnGoesFwdOnly := #MultiTurnGoesFwdOnly,
                         SET_SPD_ABS := #SET_SPD_ABS,
                         POS := #MY_POS,
                         TARGET := #MASTER_POS,
                         par_lim_fwd := #par_lim_fwd,
                         par_lim_rev := #par_lim_rev,
                         par_speed_absmax := #par_speed_absmax,
                         par_dist_absmax := #par_dist_absmax,
                         par_speed_crawl := #par_speed_crawl,
                         par_dist_crawl := #par_dist_crawl,
                         par_dist_stop := #par_dist_stop,
                         speed_dir => #speed_target,
                         ER => #ER_SET2,
                         ER_W => #ER_W);
END_REGION

REGION Network 4 (SCL)
   #delta_pos := LIMIT(IN := #MASTER_POS - #MY_POS, MN := - #par_max_Pos_delta, MX := #par_max_Pos_delta);

   IF (NOT #ER_SET) THEN
       #speed_cor := #par_max_Vcor * #delta_pos / #par_max_Pos_delta;
   ELSE
       #speed_cor := 0;
   END_IF;
END_REGION

REGION Network 5 (SCL)
   #set_speed_substantial := ABS(#SET_SPD) > #parSpeedMinThreshold;
   #set_speed_miniscule := NOT #set_speed_substantial;


   #delta:=ABS(#MY_POS - #MASTER_POS);
   #in_vicinity := #delta < #par_prec_auto;

   IF (#set_speed_substantial) THEN
       #temp_speed := #SET_SPD + #speed_cor;
   ELSE
       #temp_speed := #speed_target;
   END_IF;

   IF #set_speed_substantial OR NOT #in_vicinity THEN
       #should_move := true;
   END_IF;
   IF #set_speed_miniscule AND #speed_target = 0 THEN
       #should_move := false;
   END_IF;


   IF (#should_move) THEN
       #SPEED_OUT := #temp_speed;
   ELSE
       #SPEED_OUT := 0;
   END_IF;
END_REGION
END_FUNCTION

FUNCTION "mot_speed_by_target" : Void   // FC7, FBD
{ S7_Optimized_Access := 'TRUE' }
VERSION : 0.1
// stored: AutoNumber true, IsIECCheckEnabled false, SetENOAutomatically false, UDAEnableTagReadback false
   VAR_INPUT
      isMultiturn : Bool;
      MultiTurnGoesFwdOnly : Bool;
      SET_SPD_ABS : Real;
      POS : Real;
      TARGET : Real;
      par_lim_fwd : Real;
      par_lim_rev : Real;
      par_speed_absmax : Real;
      par_dist_absmax : Real;
      par_speed_crawl : Real;
      par_dist_crawl : Real;
      par_dist_stop : Real;
   END_VAR
   VAR_OUTPUT
      speed_dir : Real;
      ER : Bool;
      ER_W : WString;
   END_VAR
   VAR_TEMP
      target_plus_TURN : Real;
      target_minus_TURN : Real;
      target_local : Real;
      dir_fwd : Bool;
      dir_rev : Bool;
      speed_fwd : Real;
      speed_rev : Real;
      set_spd_w_dir : Real;
      turn : Real;
      dist_to_target : Real;
      dist_to_target_plus_turn : Real;
      dist_to_target_minus_turn : Real;
      distance1 : Real;
      distance2plus : Real;
      turn_inv : Real;
      distance3minus : Real;
      closest0 : Bool;
      closest1Plus : Bool;
      closest2Minus : Bool;
      target_normal : Real;
   END_VAR
BEGIN

REGION Network 2 (SCL)
   IF "ER_0_root".ACK THEN
       #ER_W := WSTRING#'';
       #ER := false;

   END_IF;
   #turn := #par_lim_fwd - #par_lim_rev;
   #turn_inv := - #turn;
END_REGION

REGION Network 3
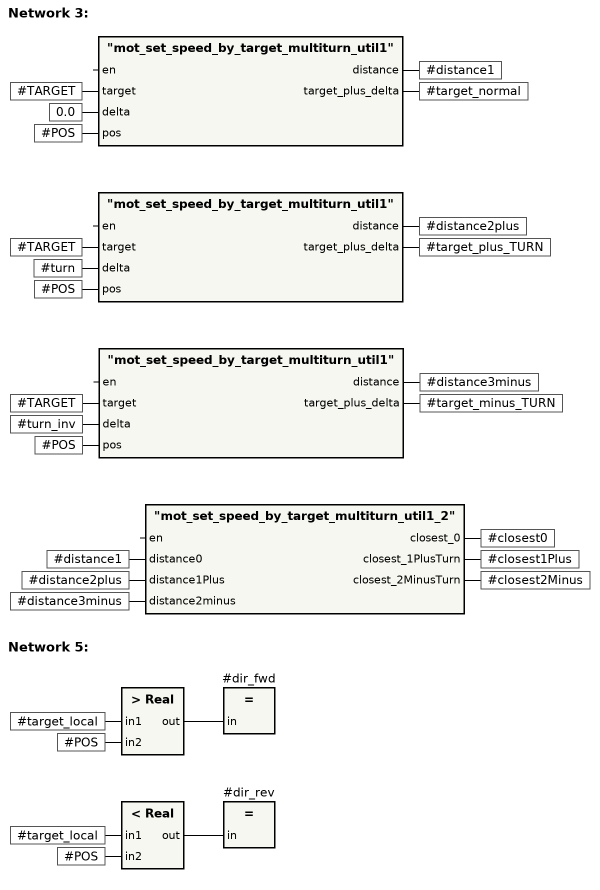
   "mot_set_speed_by_target_multiturn_util1"(target := #TARGET,
                           delta := 0.0,
                           pos := #POS,
                           distance => #distance1,
                           target_plus_delta => #target_normal);
   "mot_set_speed_by_target_multiturn_util1"(target := #TARGET,
                           delta := #turn,
                           pos := #POS,
                           distance => #distance2plus,
                           target_plus_delta => #target_plus_TURN);
   "mot_set_speed_by_target_multiturn_util1"(target := #TARGET,
                           delta := #turn_inv,
                           pos := #POS,
                           distance => #distance3minus,
                           target_plus_delta => #target_minus_TURN);
   "mot_set_speed_by_target_multiturn_util1_2"(distance0 := #distance1,
                           distance1Plus := #distance2plus,
                           distance2minus := #distance3minus,
                           closest_0 => #closest0,
                           closest_1PlusTurn => #closest1Plus,
                           closest_2MinusTurn => #closest2Minus);
END_REGION

REGION Network 4 (SCL)
   IF #isMultiturn AND NOT #ER THEN
       IF #MultiTurnGoesFwdOnly THEN
           IF #closest1Plus THEN
               #target_local := #target_plus_TURN;
           ELSE
               #target_local := #target_normal;
           END_IF;
       ELSE
           IF #closest1Plus THEN
               #target_local := #target_plus_TURN;
           ELSIF #closest2Minus THEN
               #target_local := #target_minus_TURN;
           ELSE
               #target_local := #target_normal;
           END_IF;
       END_IF;


   ELSE
       #target_local := #TARGET;
   END_IF;
END_REGION

REGION Network 5
   #dir_fwd := #target_local > #POS;
   #dir_rev := #target_local < #POS;
END_REGION

REGION Network 6
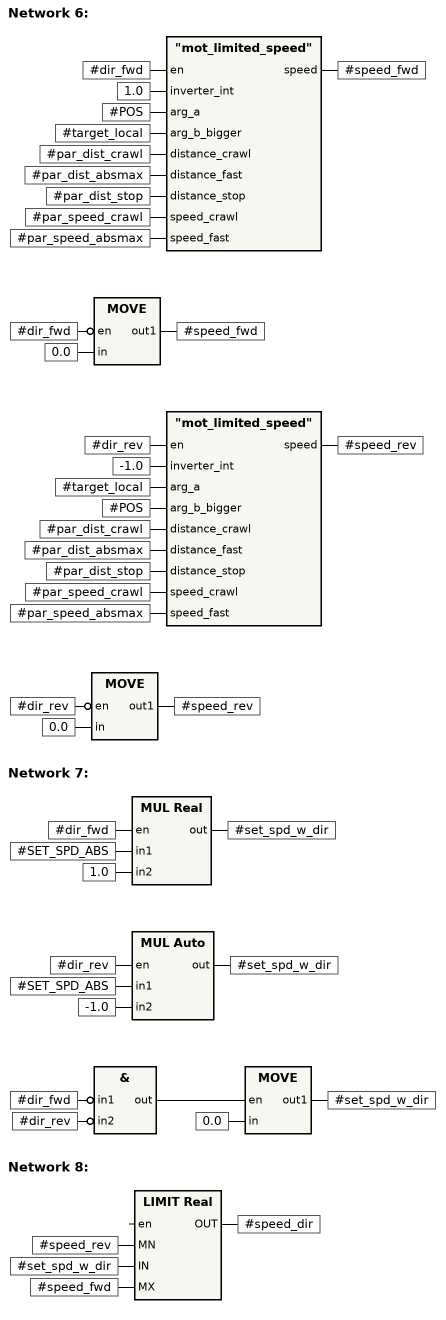
   IF #dir_fwd THEN
       "mot_limited_speed"(inverter_int := 1.0,
                           arg_a := #POS,
                           arg_b_bigger := #target_local,
                           distance_crawl := #par_dist_crawl,
                           distance_fast := #par_dist_absmax,
                           distance_stop := #par_dist_stop,
                           speed_crawl := #par_speed_crawl,
                           speed_fast := #par_speed_absmax,
                           speed => #speed_fwd);
   END_IF;
   IF NOT #dir_fwd THEN #speed_fwd := 0.0; END_IF;
   IF #dir_rev THEN
       "mot_limited_speed"(inverter_int := -1.0,
                           arg_a := #target_local,
                           arg_b_bigger := #POS,
                           distance_crawl := #par_dist_crawl,
                           distance_fast := #par_dist_absmax,
                           distance_stop := #par_dist_stop,
                           speed_crawl := #par_speed_crawl,
                           speed_fast := #par_speed_absmax,
                           speed => #speed_rev);
   END_IF;
   IF NOT #dir_rev THEN #speed_rev := 0.0; END_IF;
END_REGION

REGION Network 7
   IF #dir_fwd THEN #set_spd_w_dir := #SET_SPD_ABS * 1.0; END_IF;
   IF #dir_rev THEN #set_spd_w_dir := #SET_SPD_ABS * (-1.0); END_IF;
   IF NOT #dir_fwd AND NOT #dir_rev THEN #set_spd_w_dir := 0.0; END_IF;
END_REGION

REGION Network 8
   #speed_dir := LIMIT(MN := #speed_rev, IN := #set_spd_w_dir, MX := #speed_fwd);
END_REGION
END_FUNCTION

FUNCTION "mot_set_speed_by_target_multiturn_util1" : Void   // FC23, FBD
{ S7_Optimized_Access := 'TRUE' }
VERSION : 0.1
// stored: AutoNumber true, IsIECCheckEnabled false, SetENOAutomatically false, UDAEnableTagReadback false
   VAR_INPUT
      target : Real;
      delta : Real;
      pos : Real;
   END_VAR
   VAR_OUTPUT
      distance : Real;
      target_plus_delta : Real;
   END_VAR
BEGIN

REGION Network 2 (SCL)
   #target_plus_delta := #target + #delta
   ;
END_REGION

REGION Network 3 (SCL)
   #distance:= ABS(#target_plus_delta - #pos);
END_REGION
END_FUNCTION

FUNCTION "mot_set_speed_by_target_multiturn_util1_2" : Void   // FC24, FBD
{ S7_Optimized_Access := 'TRUE' }
VERSION : 0.1
// stored: AutoNumber true, IsIECCheckEnabled false, SetENOAutomatically false, UDAEnableTagReadback false
   VAR_INPUT
      distance0 : Real;
      distance1Plus : Real;
      distance2minus : Real;
   END_VAR
   VAR_OUTPUT
      closest_0 : Bool;
      closest_1PlusTurn : Bool;
      closest_2MinusTurn : Bool;
   END_VAR
BEGIN

REGION Network 1 (SCL)
   #closest_0 := #closest_1PlusTurn := #closest_2MinusTurn := false;

   IF #distance0 <= #distance1Plus AND #distance0 <= #distance2minus THEN
       #closest_0 := true;
   ELSIF #distance1Plus <= #distance0 AND #distance1Plus <= #distance2minus THEN
       #closest_1PlusTurn := true;
   ELSE
       #closest_2MinusTurn := true;
   END_IF;
END_REGION
END_FUNCTION

FUNCTION "mot_limited_speed" : Void   // FC12, FBD
{ S7_Optimized_Access := 'TRUE' }
VERSION : 0.1
// stored: AutoNumber true, IsIECCheckEnabled false, SetENOAutomatically false, UDAEnableTagReadback false
   VAR_INPUT
      inverter_int : Real;
      arg_a : Real;
      arg_b_bigger : Real;
      distance_crawl : Real;
      distance_fast : Real;
      distance_stop : Real;
      speed_crawl : Real;
      speed_fast : Real;
   END_VAR
   VAR_OUTPUT
      speed : Real;
   END_VAR
   VAR_TEMP
      distance1 : Real;
      distance : Real;
      can_stop : Bool;
      norm : Real;
      speed_bef_inver : Real;
   END_VAR
BEGIN

REGION Network 1
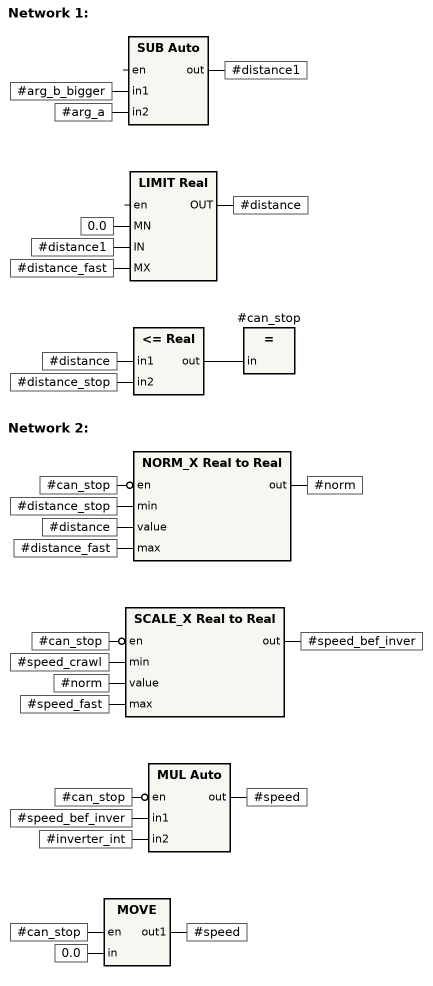
   #distance1 := #arg_b_bigger - #arg_a;
   #distance := LIMIT(MN := 0.0, IN := #distance1, MX := #distance_fast);
   #can_stop := #distance <= #distance_stop;
END_REGION

REGION Network 2
   IF NOT #can_stop THEN
       #norm := NORM_X(MIN := #distance_stop, VALUE := #distance, MAX := #distance_fast);
       #speed_bef_inver := SCALE_X(MIN := #speed_crawl, VALUE := #norm, MAX := #speed_fast);
       #speed := #speed_bef_inver * #inverter_int;
   END_IF;
   IF #can_stop THEN #speed := 0.0; END_IF;
END_REGION
END_FUNCTION

FUNCTION "mot_speed_by_pos" : Void   // FC10, FBD
{ S7_Optimized_Access := 'TRUE' }
VERSION : 0.1
// stored: AutoNumber true, IsIECCheckEnabled false, SetENOAutomatically false, UDAEnableTagReadback false
   VAR_INPUT
      SET_SPD_DIR : Real;
      POS : Real;
      xFwdOk : Bool;
      xRevOk : Bool;
      par_fwd_limit : Real;
      par_rev_limit : Real;
      par_dist_fast : Real;
      par_speed_fast : Real;
      par_dist_crawl : Real;
      par_speed_crawl : Real;
      par_dist_stop : Real;
   END_VAR
   VAR_OUTPUT
      speed_dir : Real;
   END_VAR
   VAR_TEMP
      speed_limited_fwd : Real;
      speed_limited_rev : Real;
   END_VAR
BEGIN

REGION Network 2
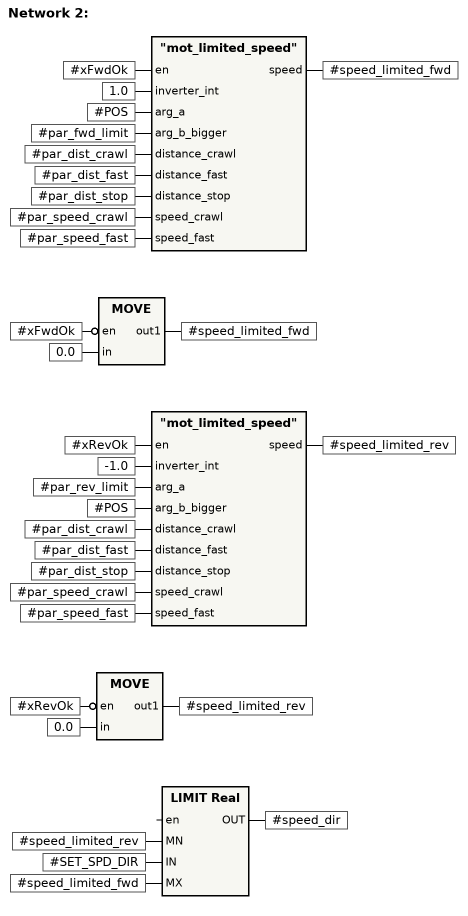
   IF #xFwdOk THEN
       "mot_limited_speed"(inverter_int := 1.0,
                           arg_a := #POS,
                           arg_b_bigger := #par_fwd_limit,
                           distance_crawl := #par_dist_crawl,
                           distance_fast := #par_dist_fast,
                           distance_stop := #par_dist_stop,
                           speed_crawl := #par_speed_crawl,
                           speed_fast := #par_speed_fast,
                           speed => #speed_limited_fwd);
   END_IF;
   IF NOT #xFwdOk THEN #speed_limited_fwd := 0.0; END_IF;
   IF #xRevOk THEN
       "mot_limited_speed"(inverter_int := -1.0,
                           arg_a := #par_rev_limit,
                           arg_b_bigger := #POS,
                           distance_crawl := #par_dist_crawl,
                           distance_fast := #par_dist_fast,
                           distance_stop := #par_dist_stop,
                           speed_crawl := #par_speed_crawl,
                           speed_fast := #par_speed_fast,
                           speed => #speed_limited_rev);
   END_IF;
   IF NOT #xRevOk THEN #speed_limited_rev := 0.0; END_IF;
   #speed_dir := LIMIT(MN := #speed_limited_rev, IN := #SET_SPD_DIR, MX := #speed_limited_fwd);
END_REGION
END_FUNCTION

FUNCTION_BLOCK "auto_analog_NORMAL"   // FB5, FBD
{ S7_Optimized_Access := 'TRUE' }
VERSION : 0.1
// stored: AutoNumber true, IsIECCheckEnabled false, IsRetainMemResEnabled false, MemoryReserve 100, SetENOAutomatically false, UDAEnableTagReadback false
   VAR_INPUT
      ALLOWED : Bool;
      MultiTurnGoesFwdOnly : Bool;
      isMultiturn : Bool;
      arrived_missed : Bool;
      SET_SPD_ABS : Real;
      POS : Real;
      TARGET : Real;
      FOLLOW : Bool;
      xFwdOK : Bool;
      xRevOK : Bool;
      par_spd_absmax : Real;
      par_dist_absMax : Real;
      par_spd_crawl : Real;
      par_dist_crawl : Real;
      par_dist_stop : Real;
      par_lim_fwd : Real;
      par_lim_rev : Real;
      par_prec_au : Real;
      par_tout_follw : Time;
      par_t_acc : Real;
   END_VAR
   VAR_OUTPUT
      SPEED : Real;
      INPOS : Bool;
      ER_follow : Bool;
      ER_settings : Bool;
      ER : Bool;
      erws : WString;
   END_VAR
   VAR
      SET_SPD_ABS_slowlyaccelerated { ExternalAccessible := 'False'; ExternalVisible := 'False'; ExternalWritable := 'False'} : Real;
      should_go { ExternalAccessible := 'False'; ExternalVisible := 'False'; ExternalWritable := 'False'} : Bool;
      mot_speed_slowly_accelerated_Instance { S7_SetPoint := 'True'} : "mot_speed_abs_slowly_accelerated";
      mot_speed_wdir_slowly_accelerated_Instance { S7_SetPoint := 'True'} : "mot_speed_wdir_slowly_accelerated";
      arrived1 { S7_SetPoint := 'True'} : "mot_auto_calc_arrivedFB";
      arrived2 { S7_SetPoint := 'True'} : "mot_auto_calc_arrivedFB";
      arrived3 { S7_SetPoint := 'True'} : "mot_auto_calc_arrivedFB";
      IEC_Timer_0_Instance { S7_SetPoint := 'True'} : TOF_TIME;
   END_VAR
   VAR_TEMP
      dir_fwd : Bool;
      dir_rev : Bool;
      arrived : Bool;
      speed_calculated : Real;
      speed_limited_fwd : Real;
      speed_limited_rev : Real;
      distance : Real;
      speed_limited_by_target_slowlychanging : Real;
      speed_limited_by_target : Real;
      estop_ok_no_err : Bool;
      speed_calc_abs : Real;
      speed_w_direction : Real;
      stop_now : Bool;
      ER_w : WString;
      length : Real;
      delta : Real;
      delta_minus : Real;
   END_VAR
   VAR CONSTANT
      erws_noer : WString := WSTRING#'';
      erws_1 : WString := WSTRING#'stuck fwd';
      erws_2 : WString := WSTRING#'stuck rev';
      erws_5 : WString := WSTRING#'->+';
      erws_4 : WString := WSTRING#'fast<0';
      erws_3 : WString := WSTRING#'fst<slo';
      erws_6 : WString := WSTRING#'tOUT<=0';
   END_VAR
   VAR_TEMP   // added for the SCL form of the ladder/FBD networks
      _w1 : Bool;
      _w2 : Bool;
      _w3 : Bool;
      _w4 : Bool;
   END_VAR
BEGIN

REGION Network 1
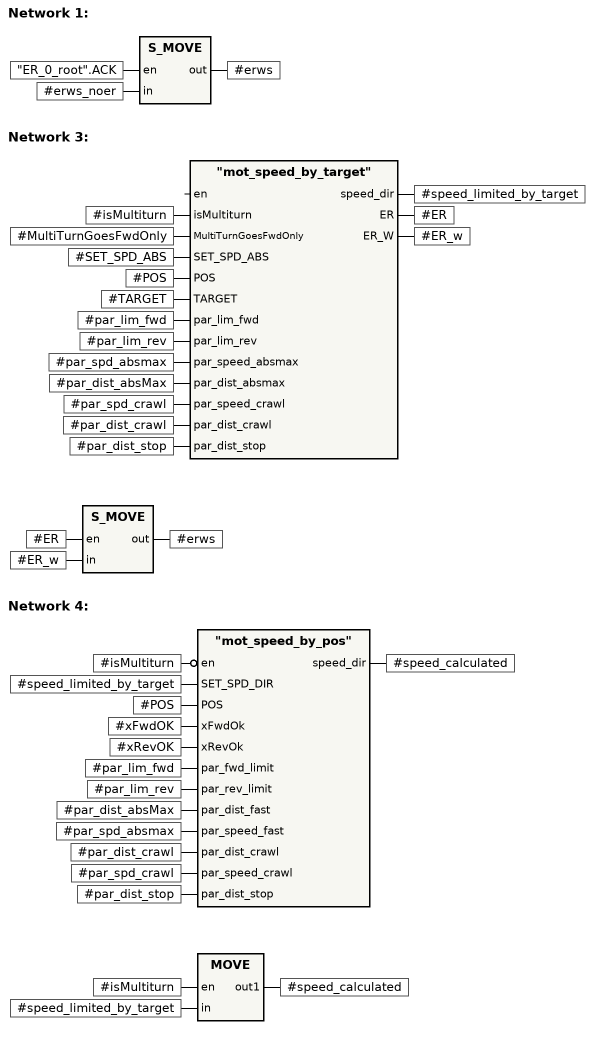
   IF "ER_0_root".ACK THEN #erws := #erws_noer; END_IF;
END_REGION

REGION Network 3
   "mot_speed_by_target"(isMultiturn := #isMultiturn,
                         MultiTurnGoesFwdOnly := #MultiTurnGoesFwdOnly,
                         SET_SPD_ABS := #SET_SPD_ABS,
                         POS := #POS,
                         TARGET := #TARGET,
                         par_lim_fwd := #par_lim_fwd,
                         par_lim_rev := #par_lim_rev,
                         par_speed_absmax := #par_spd_absmax,
                         par_dist_absmax := #par_dist_absMax,
                         par_speed_crawl := #par_spd_crawl,
                         par_dist_crawl := #par_dist_crawl,
                         par_dist_stop := #par_dist_stop,
                         speed_dir => #speed_limited_by_target,
                         ER => #ER,
                         ER_W => #ER_w);
   IF #ER THEN #erws := #ER_w; END_IF;
END_REGION

REGION Network 4
   IF NOT #isMultiturn THEN
       "mot_speed_by_pos"(SET_SPD_DIR := #speed_limited_by_target,
                          POS := #POS,
                          xFwdOk := #xFwdOK,
                          xRevOk := #xRevOK,
                          par_fwd_limit := #par_lim_fwd,
                          par_rev_limit := #par_lim_rev,
                          par_dist_fast := #par_dist_absMax,
                          par_speed_fast := #par_spd_absmax,
                          par_dist_crawl := #par_dist_crawl,
                          par_speed_crawl := #par_spd_crawl,
                          par_dist_stop := #par_dist_stop,
                          speed_dir => #speed_calculated);
   END_IF;
   IF #isMultiturn THEN #speed_calculated := #speed_limited_by_target; END_IF;
END_REGION

REGION Network 5
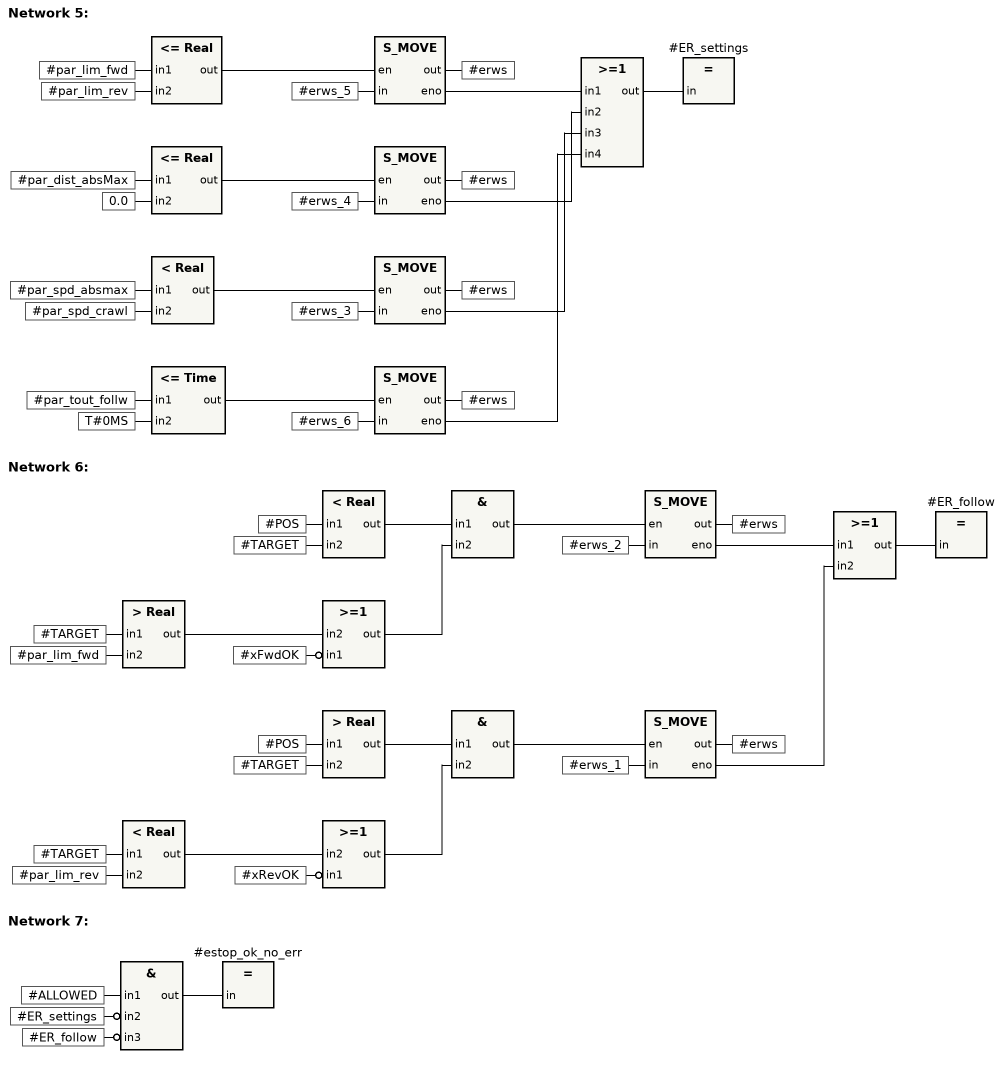
   #_w1 := #par_lim_fwd <= #par_lim_rev;
   IF #_w1 THEN #erws := #erws_5; END_IF;
   #_w2 := #par_dist_absMax <= 0.0;
   IF #_w2 THEN #erws := #erws_4; END_IF;
   #_w3 := #par_spd_absmax < #par_spd_crawl;
   IF #_w3 THEN #erws := #erws_3; END_IF;
   #_w4 := #par_tout_follw <= T#0MS;
   IF #_w4 THEN #erws := #erws_6; END_IF;
   #ER_settings := #_w1 OR #_w2 OR #_w3 OR #_w4;
END_REGION

REGION Network 6
   #_w1 := (#POS < #TARGET) AND ((#TARGET > #par_lim_fwd) OR NOT #xFwdOK);
   IF #_w1 THEN #erws := #erws_2; END_IF;
   #_w2 := (#POS > #TARGET) AND ((#TARGET < #par_lim_rev) OR NOT #xRevOK);
   IF #_w2 THEN #erws := #erws_1; END_IF;
   #ER_follow := #_w1 OR #_w2;
END_REGION

REGION Network 7
   #estop_ok_no_err := #ALLOWED AND NOT #ER_settings AND NOT #ER_follow;
END_REGION

REGION Network 8 (SCL)
   IF #isMultiturn THEN
       #length := ABS(#par_lim_fwd - #par_lim_rev);
       #delta := #length;
   ELSE
       #delta := 0    ;
   END_IF;
   #delta_minus := -#delta;
END_REGION

REGION Network 9
